INTERFACE I_DeserializerArrayForwardEnumerator EXTENDS I_Disposable

PROPERTY PUBLIC Current : I_Deserializer
GET
END_GET
END_PROPERTY

PROPERTY Index : DINT
GET
END_GET
END_PROPERTY

PROPERTY IsValid : BOOL
GET
END_GET
END_PROPERTY

METHOD MoveNext : BOOL
VAR_INPUT
END_VAR
END_METHOD

END_INTERFACE

(* stored: Version 1.1.0.1, ProductVersion 3.1.4024.12
   Itf I_DeserializerArrayForwardEnumerator: Id {5026e20b-c7dd-03e9-027c-ac6037fe2766}
   Property Current: Id {e1a5ccd4-f999-0063-237e-9476dceef8e5}
   Get Get: Id {c51d0fd0-92d2-0db5-3369-2d02f9596d49}
   Property Index: Id {62c60b3a-ddad-091d-1690-e27b9fe15a25}
   Get Get: Id {a646d3a4-edb0-0a01-3278-4685cfc39575}
   Property IsValid: Id {f3e59b95-db62-0300-22c0-31210d8eb811}
   Get Get: Id {a0cc5345-a1b2-0aba-0720-4e1ec3a1fbab}
   Method MoveNext: Id {80c8289c-517d-0a06-29e5-5b15a4e8b719} *)
